// TIA Portal V17 export
// export: Created 2025-06-26T07:49:13.0648224Z, ExportSetting WithDefaults, DisplayName Totally Integrated Automation Portal, DisplayVersion V17 Update 8, DisplayName TIA Portal Openness, DisplayVersion V17 Update 8, DisplayName TIA Portal Version Control Interface, DisplayVersion V17, DisplayName STEP 7 Professional, DisplayVersion V17 Update 8, DisplayName STEP 7 Safety, DisplayVersion V17 Update 6, DisplayName WinCC Advanced, DisplayVersion V17 Update 8
FUNCTION_BLOCK "CAN-Communication"   // FB8, FBD
{ S7_Optimized_Access := 'TRUE' }
VERSION : 0.1
// stored: AutoNumber true, IsIECCheckEnabled false, IsRetainMemResEnabled false, MemoryReserve 100, SetENOAutomatically false, UDAEnableTagReadback false
   VAR_IN_OUT
      "CAN-IDs_ToSend" : Array[0..74] of Int;
   END_VAR
   VAR
      SendBusy : Bool;
      UseFixedPoint : Bool;   // Send data on CAN as fixed point
      Memory : DInt;
      CycleCheck : Bool;
      TESTUINT_CTRL { ExternalAccessible := 'False'; ExternalVisible := 'False'; ExternalWritable := 'False'} : UInt;
      TESTUINT_SEND : UInt;
      TESTUINT_RCV : UInt;
      TOF_SendError { S7_SetPoint := 'True'} : TOF_TIME;
      CountSendAll : UDInt;
      ScaleFactor : Real := 1000.0;   // Fixed point scale factor
   END_VAR
   VAR_TEMP
      i : Int;
      UpperBound : DInt;
      NumberOfFrames : SInt;
      TestUint : UInt;
   END_VAR
BEGIN

REGION Network 1: CAN Control
   // process a CAN_CTRL command (if requested)
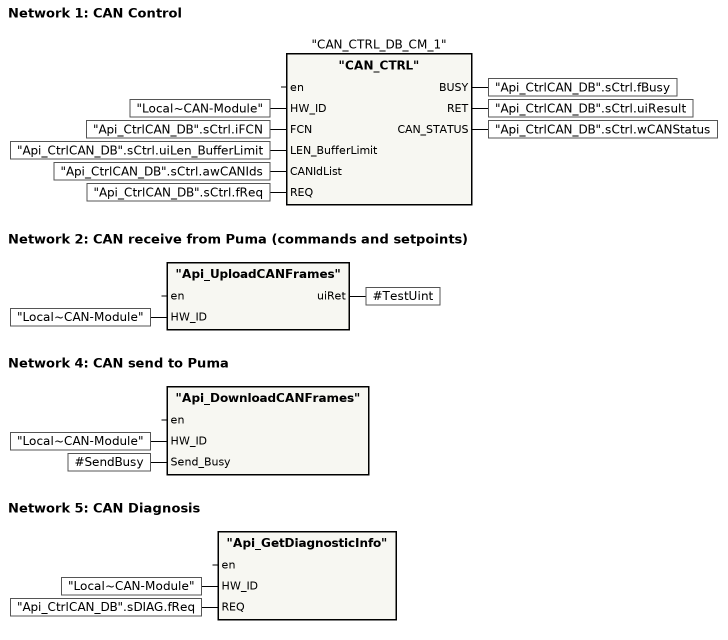
   "CAN_CTRL_DB_CM_1"(HW_ID := "Local~CAN-Module",   // "CAN_CTRL"
                      FCN := "Api_CtrlCAN_DB".sCtrl.iFCN,
                      LEN_BufferLimit := "Api_CtrlCAN_DB".sCtrl.uiLen_BufferLimit,
                      CANIdList := "Api_CtrlCAN_DB".sCtrl.awCANIds,
                      REQ := "Api_CtrlCAN_DB".sCtrl.fReq,
                      BUSY => "Api_CtrlCAN_DB".sCtrl.fBusy,
                      RET => "Api_CtrlCAN_DB".sCtrl.uiResult,
                      CAN_STATUS => "Api_CtrlCAN_DB".sCtrl.wCANStatus);
END_REGION

REGION Network 2: CAN receive from Puma (commands and setpoints)
   // function processes the upload of CAN frames and processes the uploaded CAN frames
   "Api_UploadCANFrames"(HW_ID := "Local~CAN-Module", uiRet => #TestUint);
END_REGION

REGION Network 3 (SCL): Send CAN frame select
   // The CAN SEND block can only send 19 frames each call. So every call, other frame IDs gets written into the output list.
   // HW_ID := "Local~CAN-Module"
   //Diagnosis to store error messages from CAN functions
   IF "Api_CtrlCAN_DB".sCtrl.uiResult <> 0 THEN
       #TESTUINT_CTRL:="Api_CtrlCAN_DB".sCtrl.uiResult;
   END_IF;
   IF "Api_CtrlCAN_DB".sSEND.sDemo.sDownload.uiResult <> 0 THEN
       #TESTUINT_SEND:="Api_CtrlCAN_DB".sSEND.sDemo.sDownload.uiResult;
   END_IF;
   IF #TestUint <> 0 THEN
       #TESTUINT_RCV := #TestUint;
   END_IF;

   IF NOT "Api_CtrlCAN_DB".sRCV.fReq THEN // Was ist das und wofür?
       "Api_CtrlCAN_DB".sCtrl.fReq := True;
       "Api_CtrlCAN_DB".sCtrl.iFCN := 1;
       "Api_CtrlCAN_DB".sRCV.fReq := True;
   END_IF;


   //Update current status
   IF "Api_CtrlCAN_DB".sSEND.fTransfer AND #SendBusy THEN //If completed transmission pending then check current status
       "Api_DownloadCANFrames"(HW_ID := "Local~CAN-Module",
                               Send_Busy := #SendBusy);
   END_IF; // "Api_CtrlCAN_DB".sSEND.fTransfer THEN 

   //Write IDs to send list
   IF NOT "Api_CtrlCAN_DB".sSEND.fTransfer AND NOT #SendBusy THEN // OR NOT "Api_CtrlCAN_DB".sSEND.sDemo.sRequest.fReq THEN
       // In Transfere is ready or actually no send request (first or due to error)    
       // Currently in case of error we do not resend this on, but proceed with the other ones. It is only retransmitted within the normal procedure after a complete cycle.
       // "Api_CtrlCAN_DB".sSEND.sDemo.sRequest.fError ist die error flag

       //#UpperBound := UPPER_BOUND(ARR := #"CAN-IDs_ToSend", DIM := 1);     //Upper bound of all CAN-IDs to send
       #UpperBound := 69;
       #NumberOfFrames := 0;                                               //Resetting CAN frame counter
       FOR #i := 0 TO 18 DO                                                //Writing all 10/19 CAN_IDs to send into output array
           IF #Memory + #i <= #UpperBound THEN                             //Check if there are CAN-IDs left
               "Api_CtrlCAN_DB".sSEND.sDemo.sRequest.aiCAN_ID[#i] := #"CAN-IDs_ToSend"[#i + #Memory];      //The next ID gets written into send list
               #NumberOfFrames := #NumberOfFrames + 1;                     //Count up on each frame
           ELSE
               "Api_CtrlCAN_DB".sSEND.sDemo.sRequest.aiCAN_ID[#i] := 0;    //No ID left
           END_IF;

       END_FOR;

       "Api_CtrlCAN_DB".sSEND.sDemo.sRequest.siNoFrames := #NumberOfFrames;//Send number of CAN-IDs to send to maximum (19 [0..18])
       "Api_CtrlCAN_DB".sSEND.sDemo.sRequest.fReq := TRUE;                 //send new frame if not busy

       #Memory := #Memory + #NumberOfFrames;                               //Next cycle the Next 19 IDs gets send 
       IF #Memory > #UpperBound THEN   //if all IDs got send, all gets send again
           #Memory := 0;               //Start with ID 0
           #CountSendAll += 1;
       END_IF; // IF #Memory > #UpperBound THEN

   END_IF; // IF NOT "Api_CtrlCAN_DB".sSEND.fTransfer OR NOT "Api_CtrlCAN_DB".sSEND.sDemo.sRequest.fReq THEN
END_REGION

REGION Network 4: CAN send to Puma
   // function checks if CAN frames shall be transitted, which CAN frames shall be transmitted, enters the requested CAN frames in the data field that will be written to the CM module and processes the download to the CM module
   "Api_DownloadCANFrames"(HW_ID := "Local~CAN-Module", Send_Busy := #SendBusy);
END_REGION

REGION Network 5: CAN Diagnosis
   // process "Get Diagnostic Information" (if requested)
   "Api_GetDiagnosticInfo"(HW_ID := "Local~CAN-Module", REQ := "Api_CtrlCAN_DB".sDIAG.fReq);
END_REGION

REGION Network 6: Error message via CAN
   // WinCC Alarm 3001 triggered from:
   // "CAN_Data_DB".InputData.CAN_ID_101h.Error_CAN
   // Plumb this in on the PUT side
END_REGION

REGION Network 7 (SCL): Error while sending CAN frames
   #TOF_SendError(IN:=#TESTUINT_SEND<>0,
                  PT:=T#10s);

   #TESTUINT_SEND := 0; //Reset Error

   //"WinCC_Alarm"(TriggerBit := #TOF_SendError.Q,
   //        Message := "DB_WinCCAlarms".Messages."3-Communication"."3002_ErrorWhileCANSending");
END_REGION

REGION Network 8 (SCL): Reset CAN module (queue)
   // This function resets the CAN-Module. For example sometimes the output queue for CAN-frames is full and sends an error. And the reset clears this queue, too.
   // Copied from process PLC
   IF "DB_Puma"."CAN-Reset_Required" THEN
       "Api_CtrlCAN_DB".sCtrl.fReq := True;
       "Api_CtrlCAN_DB".sCtrl.iFCN := 5;
       "DB_Puma"."CAN-Reset_Required" := FALSE;
   ELSIF "Api_CtrlCAN_DB".sCtrl.iFCN = 5 THEN

       "Api_CtrlCAN_DB".sCtrl.fReq := True;
       "Api_CtrlCAN_DB".sCtrl.iFCN := 1;
   END_IF;
END_REGION
END_FUNCTION_BLOCK
